(* Logix 5000 project; controller Add_On_MIG Emulate 5570 rev 33.11; software revision 33.00 *)

TASK MainTask (continuous, watchdog 500 ms) : MainProgram, Model

MODULES
   Local : Emulate 5570 (ICP 2, rev 33.11)
       : 1756-IB16 (ICP 3, rev 3.1, Input RPI 20 ms)
       : vendor 1 type 7 code 16 (ICP 4, rev 3.1, Output RPI 20 ms)
END_MODULES

PROGRAM MainProgram   (* main routine MainRoutine *)

ROUTINE MainRoutine   (* ladder *)
   0: ;
   1: ;
END_ROUTINE
END_PROGRAM

PROGRAM Model   (* main routine Emulation *)
VAR
   Welder1_End : BOOL;
   Welder1_Fault_Arc : BOOL;
   Welder1_Fault_Wire : BOOL;
   Welder1_Start : BOOL;
   Welder2_End : BOOL;
   Welder2_Fault_Arc : BOOL;
   Welder2_Fault_Wire : BOOL;
   Welder2_Start : BOOL;
END_VAR

ROUTINE Emulation   (* ladder *)
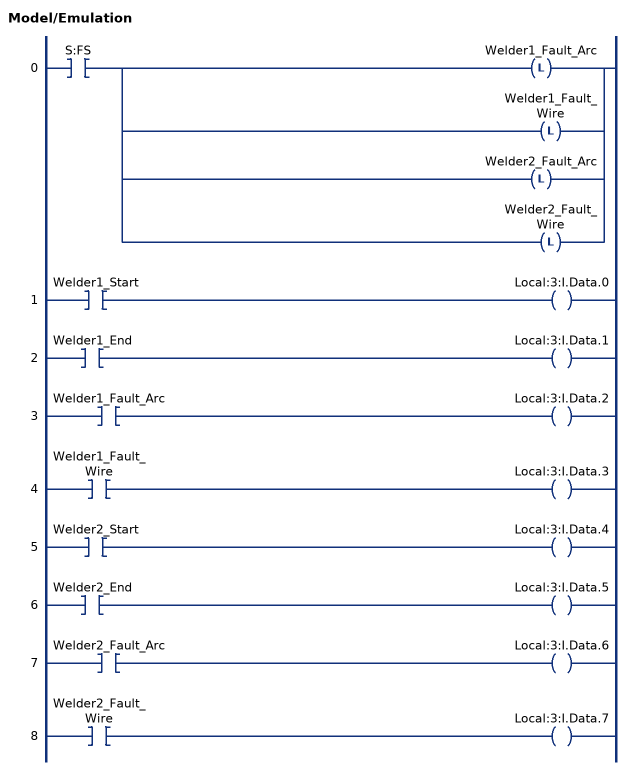
   0: XIC(S:FS)[OTL(Welder1_Fault_Arc) ,OTL(Welder1_Fault_Wire) ,OTL(Welder2_Fault_Arc) ,OTL(Welder2_Fault_Wire) ];
   1: XIC(Welder1_Start)OTE(Local:3:I.Data.0);
   2: XIC(Welder1_End)OTE(Local:3:I.Data.1);
   3: XIC(Welder1_Fault_Arc)OTE(Local:3:I.Data.2);
   4: XIC(Welder1_Fault_Wire)OTE(Local:3:I.Data.3);
   5: XIC(Welder2_Start)OTE(Local:3:I.Data.4);
   6: XIC(Welder2_End)OTE(Local:3:I.Data.5);
   7: XIC(Welder2_Fault_Arc)OTE(Local:3:I.Data.6);
   8: XIC(Welder2_Fault_Wire)OTE(Local:3:I.Data.7);
END_ROUTINE
END_PROGRAM
